(* CODESYS project CmpTemplateEventIEC.library
   Version: 3.5.8.0
   Author: 3S - Smart Software Solutions GmbH
   Title: CoDeSys Event Usage Template
   Description: Library project template with all possible element types, docu and a sample project structure
   Placeholder: PlaceholderTemplate
   DocFormat: reStructuredText
   DefaultNamespace: EVTDEMO
   LanguageModelAttribute: qualified-access-only
   Company: 3S - Smart Software Solutions GmbH

Project tree, tasks and I/O mapping:
  libraries: CAA Types Extern, * (CAA Technical Workgroup); CmpEventMgr, 3.5.8.0 (System)
  EventParameter/
    data type EVTPARAM_EvtTest
  global variables EventIDs
*)

// EventParameter/EVTPARAM_EvtTest
(**
 * <category>Event parameter</category>
 * <element name="dwParam1" type="IN">Just a test parameter, value will be 17</element>
 * <element name="xParam2" type="IN">Just another test parameter, value will be TRUE</element>
 *)
TYPE EVTPARAM_EvtTest :
STRUCT
	dwParam1: DWORD;	// a test parameter
	xParam2: BOOL;		// another test parameter
END_STRUCT
END_TYPE

// EventIDs
//{attribute 'qualified_only'}
//{attribute 'conditionalshow' := 'SomeText'}
//{attribute 'conditionalshow'}
//{attribute 'hide'}
VAR_GLOBAL CONSTANT
	// ComponentID to specify for EventOpen
	CmpId_CmpTest: DWORD := 16#2000;

	(* IDs for the event parameter structures *)
	EVTPARAMID_CmpTemplateEventIEC : WORD := 16#0001;
	EVTVERSION_CmpTemplateEventIEC : WORD := 16#0001;

	(**
	 * <category>Events</category>
	 * <description>Event is sent for test, in every runtime comm cycle</description>
	 * <param name="pEventParam" type="IN">EVTPARAM_EvtTest</param>
	 *)
	EVT_Test : DWORD := SHL(UINT_TO_DWORD(EventClass.EVTCLASS_INFO), 16) OR 16#00000001; 
END_VAR
